FUNCTION_BLOCK CrcCheck
VAR_INPUT
END_VAR
VAR_OUTPUT
END_VAR
VAR
  act_crc: UINT;
  previous_crc: UINT;
END_VAR

METHOD data_changed : BOOL
VAR_INPUT
  data_ptr: POINTER TO BYTE;
  data_size: UDINT;
END_VAR
act_crc := F_DATA_TO_CRC16_CCITT(data_ptr, data_size, 0);
data_changed := act_crc <> previous_crc;
END_METHOD

METHOD reset
VAR_INPUT
END_VAR
previous_crc := act_crc;
END_METHOD

END_FUNCTION_BLOCK

(* stored: Version 1.1.0.1, ProductVersion 3.1.4022.18
   POU CrcCheck: Id {9fc5645c-e006-4563-b398-2c69432ab599}, SpecialFunc None
   Method data_changed: Id {859b12b2-30a4-47dc-8f26-7933132f402d}
   Method reset: Id {a26de202-1f26-4a50-a38f-d7c60aa4dfe1} *)
